TEXTLIST TextList_Cryo_Relays_Parameters
  0 = '' | FR: 'Régler le seuil inférieur du 1er étage (deg Kelvin)' | EN: 'Set first stage LL (deg Kelvin)'
  1 = '' | FR: 'Régler le seuil supérieur du 1er étage (deg Kelvin)' | EN: 'Set first stage UL (deg Kelvin)'
  2 = '' | FR: 'Régler le seuil inférieur du 2ème étage (deg Kelvin)' | EN: 'Set second stage LL (deg Kelvin)'
  3 = '' | FR: 'Régler le seuil supérieur du 2ème étage (deg Kelvin)' | EN: 'Set second stage UL (deg Kelvin)'
  4 = '' | FR: 'Régler la pression inférieure du thermocouple de la cryo (microns)' | EN: 'Set Pump TC LL (microns)'
  5 = '' | FR: 'Régler la pression supérieure du thermocouple de la cryo (microns)' | EN: 'Set Pump TC UL (microns)'
  6 = '' | FR: 'Régler la pression inférieure du thermocouple auxiliaire (microns)' | EN: 'Set AUX TC LL (microns)'
  7 = '' | FR: 'Régler la pression supérieure du thermocouple auxiliaire (microns)' | EN: 'Set AUX TC UL (microns)'
  8 = '' | FR: 'Régler le temps du relais (0-9999 secondes)' | EN: 'Set time relay (0-9999 seconds)'
  10 = '' | FR: 'Activation inconditionnelle' | EN: 'Set unconditional ON'
  11 = '' | FR: 'Désactivation inconditionnelle' | EN: 'Set unconditional OFF'
  12 = '' | FR: "Régler le suivi de l'état de régénération" | EN: 'Set as REGEN status tracking relay'
  13 = '' | FR: "Régler le suivi de l'état de vanne primaire" | EN: 'Set as rough valve tracking relay'
  15 = '' | FR: "Régler le suivi de l'état de la pompe cryo" | EN: 'Set as pump motor ON/OFF status tracking relay'
  9 = '' | FR: '-' | EN: '-'
  14 = '' | FR: '-' | EN: '-'
   = ''
END_TEXTLIST

(* stored: Version 1.1.0.1, ProductVersion 3.1.4026.18
   TextList TextList_Cryo_Relays_Parameters: Id {bd13558d-6e57-4624-80f7-fb7d49db89b2} *)
